// TIA Portal V17 export
// export: Created 2025-03-05T07:59:26.3557512Z, ExportSetting WithDefaults, DisplayName Totally Integrated Automation Portal, DisplayVersion V17 Update 8, DisplayName TIA Portal Openness, DisplayVersion V17 Update 8, DisplayName TIA Portal Version Control Interface, DisplayVersion V17, DisplayName SINAMICS Startdrive Advanced, DisplayVersion V17 SP2, DisplayName SINAMICS Startdrive G110M, G120, G120C, G120D, G120P, G115D, DisplayVersion V17 SP2, DisplayName SINAMICS Startdrive G130, G150, S120, S150, SINAMICS MV, S210, DisplayVersion V17 SP2, DisplayName STEP 7 Professional, DisplayVersion V17 Update 8, DisplayName SINUMERIK ONE STEP 7 Toolbox, DisplayVersion V17 Update 12, DisplayName SINUMERIK 840D sl STEP 7 Toolbox, DisplayVersion V17 Update 12, DisplayName STEP 7 Safety, DisplayVersion V17 Update 6, DisplayName WinCC Advanced, DisplayVersion V17 Update 8
FUNCTION "FC8007_UNIT_03_PART_STATUS_FULL_DEPTH" : Void   // FC8007, LAD
{ S7_Optimized_Access := 'TRUE' }
VERSION : 0.1
// stored: AutoNumber false, IsIECCheckEnabled false, SetENOAutomatically false, UDAEnableTagReadback false
BEGIN

REGION Network 1: FIXTURE 1 PART STATUS UNIT 01
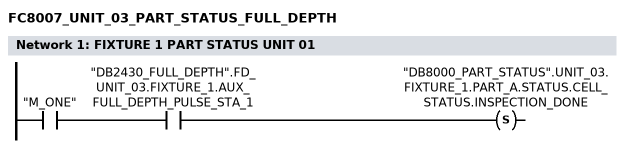
   RUNG wire#powerrail
      Contact( "M_ONE" )
      Contact( "DB2430_FULL_DEPTH".FD_UNIT_03.FIXTURE_1.AUX_FULL_DEPTH_PULSE_STA_1 )
      S_Coil( "DB8000_PART_STATUS".UNIT_03.FIXTURE_1.PART_A.STATUS.CELL_STATUS.INSPECTION_DONE )
   END_RUNG
   // the same network as SCL:
   IF "M_ONE" AND "DB2430_FULL_DEPTH".FD_UNIT_03.FIXTURE_1.AUX_FULL_DEPTH_PULSE_STA_1 THEN
       "DB8000_PART_STATUS".UNIT_03.FIXTURE_1.PART_A.STATUS.CELL_STATUS.INSPECTION_DONE := TRUE;
   END_IF;
END_REGION
END_FUNCTION
